PROGRAM MAIN
VAR
END_VAR

// To activate a section in the progem it has to be written in the MAIN (PRG). the sequence of the sections would determine what run first in the progrem.
Common_Pulses();
Pumps();
Loaders();
Alarms();
	GVL.testvar := Pumps.Pump_1.Status_Word;

END_PROGRAM

(* stored: Version 1.1.0.1, ProductVersion 3.1.4024.13
   POU MAIN: Id {54a8759e-438d-41aa-88f1-b08bf98f9189}, SpecialFunc None *)
